// TIA Portal V15.1 export
// export: Created 2020-06-12T07:35:53.7568359Z, ExportSetting None, DisplayName Totally Integrated Automation Portal, DisplayVersion V15.1, DisplayName TIA Portal Openness, DisplayVersion V15.1, DisplayName STEP 7 Professional, DisplayVersion V15.1, DisplayName STEP 7 Safety, DisplayVersion V15.1, DisplayName WinCC Advanced, DisplayVersion V15.1
FUNCTION "RCW_Pumps" : Void   // FC152, FBD
TITLE = Pumps c logic
{ S7_Optimized_Access := 'TRUE' }
// The three pumps is using with redundancy in mode 2R+1S
// stored: SetENOAutomatically False
   VAR_TEMP
      tOnM1 : Bool;
      tOnM2 : Bool;
      tOnM3 : Bool;
      tOn1 : Bool;
      tOn2 : Bool;
      tOn3 : Bool;
   END_VAR
BEGIN

REGION Network 1: Pumps redundancy
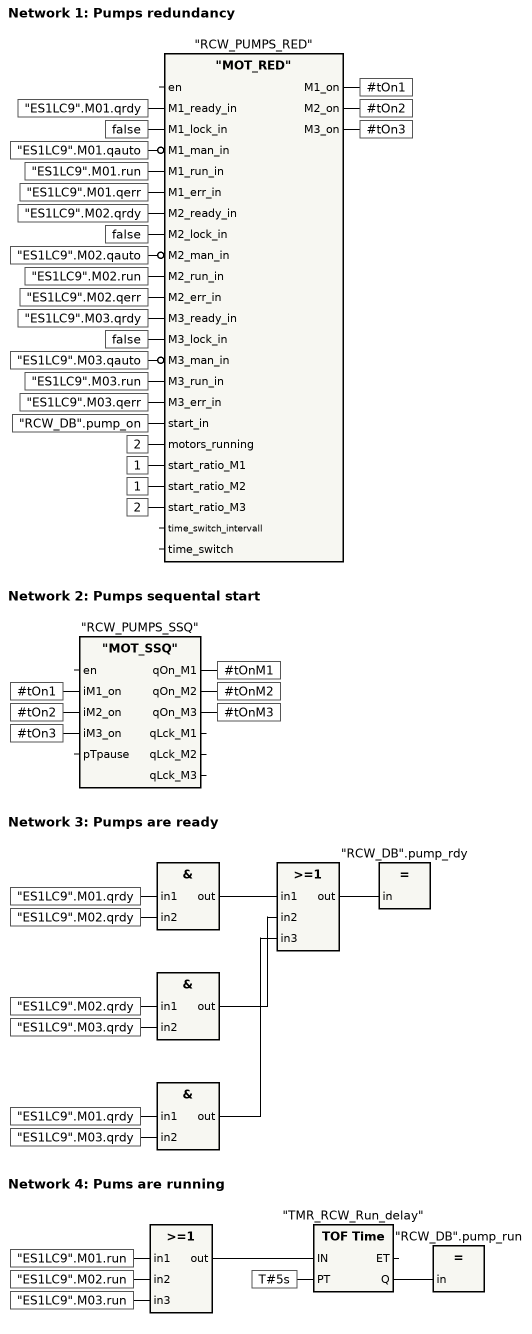
   "RCW_PUMPS_RED"(M1_ready_in := "ES1LC9".M01.qrdy,   // "MOT_RED"
                   M1_lock_in := false,
                   M1_man_in := NOT "ES1LC9".M01.qauto,
                   M1_run_in := "ES1LC9".M01.run,
                   M1_err_in := "ES1LC9".M01.qerr,
                   M2_ready_in := "ES1LC9".M02.qrdy,
                   M2_lock_in := false,
                   M2_man_in := NOT "ES1LC9".M02.qauto,
                   M2_run_in := "ES1LC9".M02.run,
                   M2_err_in := "ES1LC9".M02.qerr,
                   M3_ready_in := "ES1LC9".M03.qrdy,
                   M3_lock_in := false,
                   M3_man_in := NOT "ES1LC9".M03.qauto,
                   M3_run_in := "ES1LC9".M03.run,
                   M3_err_in := "ES1LC9".M03.qerr,
                   start_in := "RCW_DB".pump_on,
                   motors_running := 2,
                   start_ratio_M1 := 1,
                   start_ratio_M2 := 1,
                   start_ratio_M3 := 2,
                   M1_on => #tOn1,
                   M2_on => #tOn2,
                   M3_on => #tOn3);
END_REGION

REGION Network 2: Pumps sequental start
   "RCW_PUMPS_SSQ"(iM1_on := #tOn1,   // "MOT_SSQ"
                   iM2_on := #tOn2,
                   iM3_on := #tOn3,
                   qOn_M1 => #tOnM1,
                   qOn_M2 => #tOnM2,
                   qOn_M3 => #tOnM3);
END_REGION

REGION Network 3: Pumps are ready
   // at least two are ready
   "RCW_DB".pump_rdy := ("ES1LC9".M01.qrdy AND "ES1LC9".M02.qrdy) OR ("ES1LC9".M02.qrdy AND "ES1LC9".M03.qrdy) OR ("ES1LC9".M01.qrdy AND "ES1LC9".M03.qrdy);
END_REGION

REGION Network 4: Pums are running
   "TMR_RCW_Run_delay".TOF(IN := "ES1LC9".M01.run OR "ES1LC9".M02.run OR "ES1LC9".M03.run, PT := T#5s);
   "RCW_DB".pump_run := "TMR_RCW_Run_delay".Q;
END_REGION

REGION Network 5: .M01 Lock
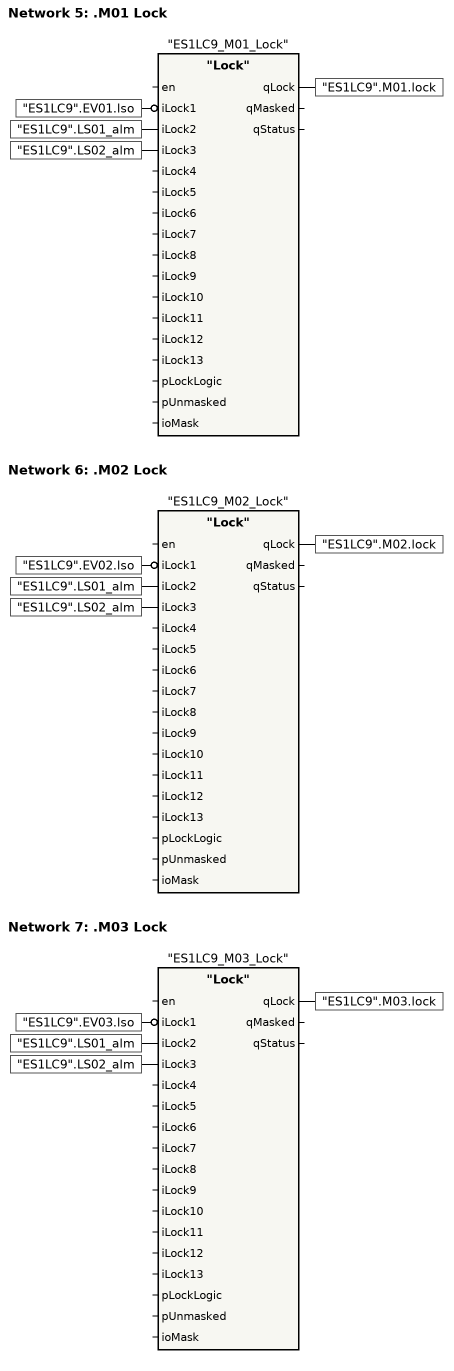
   "ES1LC9_M01_Lock"(iLock1 := NOT "ES1LC9".EV01.lso,   // "Lock"
                     iLock2 := "ES1LC9".LS01_alm,
                     iLock3 := "ES1LC9".LS02_alm,
                     qLock => "ES1LC9".M01.lock);
END_REGION

REGION Network 6: .M02 Lock
   "ES1LC9_M02_Lock"(iLock1 := NOT "ES1LC9".EV02.lso,   // "Lock"
                     iLock2 := "ES1LC9".LS01_alm,
                     iLock3 := "ES1LC9".LS02_alm,
                     qLock => "ES1LC9".M02.lock);
END_REGION

REGION Network 7: .M03 Lock
   "ES1LC9_M03_Lock"(iLock1 := NOT "ES1LC9".EV03.lso,   // "Lock"
                     iLock2 := "ES1LC9".LS01_alm,
                     iLock3 := "ES1LC9".LS02_alm,
                     qLock => "ES1LC9".M03.lock);
END_REGION

REGION Network 8: .M01 start
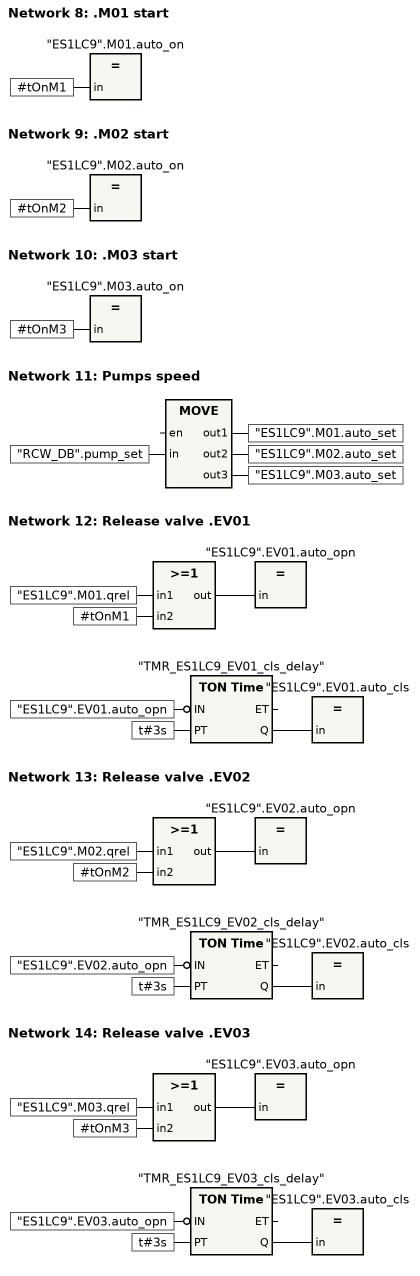
   "ES1LC9".M01.auto_on := #tOnM1;
END_REGION

REGION Network 9: .M02 start
   "ES1LC9".M02.auto_on := #tOnM2;
END_REGION

REGION Network 10: .M03 start
   "ES1LC9".M03.auto_on := #tOnM3;
END_REGION

REGION Network 11: Pumps speed
   "ES1LC9".M01.auto_set := "RCW_DB".pump_set;
   "ES1LC9".M02.auto_set := "RCW_DB".pump_set;
   "ES1LC9".M03.auto_set := "RCW_DB".pump_set;
END_REGION

REGION Network 12: Release valve .EV01
   // NR!
   "ES1LC9".EV01.auto_opn := "ES1LC9".M01.qrel OR #tOnM1;
   "TMR_ES1LC9_EV01_cls_delay".TON(IN := NOT "ES1LC9".EV01.auto_opn, PT := t#3s);
   "ES1LC9".EV01.auto_cls := "TMR_ES1LC9_EV01_cls_delay".Q;
END_REGION

REGION Network 13: Release valve .EV02
   // NR!
   "ES1LC9".EV02.auto_opn := "ES1LC9".M02.qrel OR #tOnM2;
   "TMR_ES1LC9_EV02_cls_delay".TON(IN := NOT "ES1LC9".EV02.auto_opn, PT := t#3s);
   "ES1LC9".EV02.auto_cls := "TMR_ES1LC9_EV02_cls_delay".Q;
END_REGION

REGION Network 14: Release valve .EV03
   // NR!
   "ES1LC9".EV03.auto_opn := "ES1LC9".M03.qrel OR #tOnM3;
   "TMR_ES1LC9_EV03_cls_delay".TON(IN := NOT "ES1LC9".EV03.auto_opn, PT := t#3s);
   "ES1LC9".EV03.auto_cls := "TMR_ES1LC9_EV03_cls_delay".Q;
END_REGION

REGION Network 15: Enable an alarms group #1
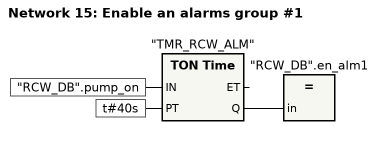
   "TMR_RCW_ALM".TON(IN := "RCW_DB".pump_on, PT := t#40s);
   "RCW_DB".en_alm1 := "TMR_RCW_ALM".Q;
END_REGION
END_FUNCTION
